Omron CX-Programmer project NuevoProyecto (CX-Programmer 9.40)

# PLC NuevoPLC1: CQM1 CPU41

## Global symbols (name address type ; comment)
A_mas 100.00 BOOL
B_mas 100.04 BOOL
B_menos 100.05 BOOL
C_mas 100.08 BOOL
C_menos 100.09 BOOL
D_mas 100.12 BOOL
Y_0 100.15 BOOL
a_0 0.00 BOOL
a_1 0.01 BOOL
b_0 0.04 BOOL
b_1 0.05 BOOL
c_0 0.08 BOOL
c_1 0.09 BOOL
pe 0.13 BOOL
pm 0.14 BOOL
pp 0.15 BOOL

## Program NuevoPrograma1 (no task)

### Section Sección1

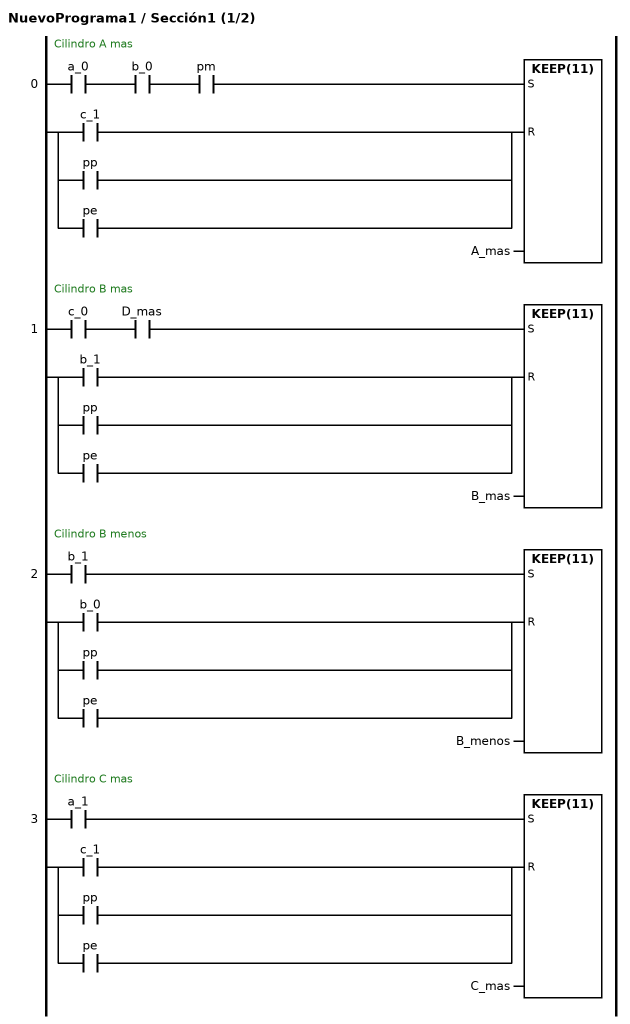
; rung 0: Cilindro A mas
LD a_0
AND b_0
AND pm
LD c_1
OR pp
OR pe
KEEP(11) A_mas
; rung 1: Cilindro B mas
LD c_0
AND D_mas
LD b_1
OR pp
OR pe
KEEP(11) B_mas
; rung 2: Cilindro B menos
LD b_1
LD b_0
OR pp
OR pe
KEEP(11) B_menos
; rung 3: Cilindro C mas
LD a_1
LD c_1
OR pp
OR pe
KEEP(11) C_mas

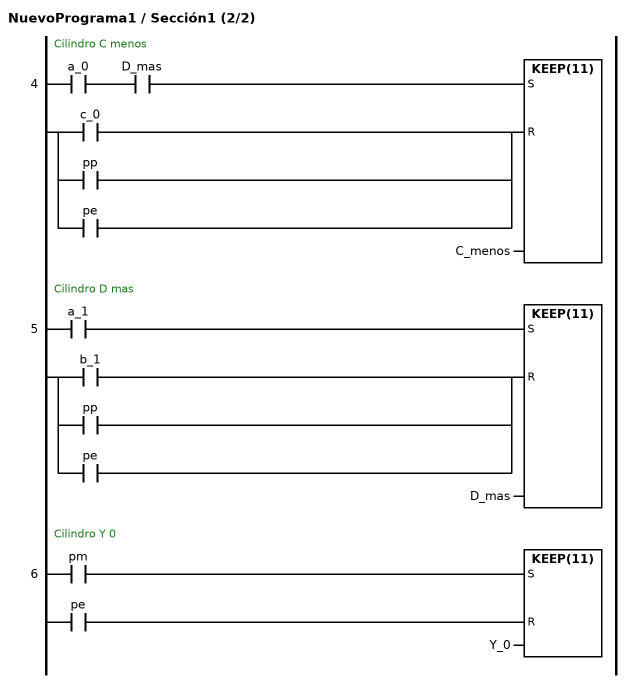
; rung 4: Cilindro C menos
LD a_0
AND D_mas
LD c_0
OR pp
OR pe
KEEP(11) C_menos
; rung 5: Cilindro D mas
LD a_1
LD b_1
OR pp
OR pe
KEEP(11) D_mas
; rung 6: Cilindro Y 0
LD pm
LD pe
KEEP(11) Y_0

### Section END
; rung 0
END(01)